// TIA Portal V20 export
FUNCTION_BLOCK "FB_Alarms_Safety"   // FB150, SCL
{ S7_Optimized_Access := 'TRUE' }
// stored: AutoNumber false, MemoryReserve 100, SetENOAutomatically false
   VAR
      sTimerEmergencyPowLaser : IEC_TIMER;
   END_VAR
BEGIN
   REGION Description header 
       //==================================================================================
       // POSALUX Swiss SA / (C) Copyright 2024
       //----------------------------------------------------------------------------------
       // Title: Affichage Alarmes/Messages Safety
       // Comment/Function: 
       //
       // Author: Michel FAIVRE
       // Engineering: TIA Portal v17
       //----------------------------------------------------------------------------------
       // Change log table:
       // Version  | Date     | Expert in charge | Changes applied
       // ---------|----------|------------------|------------------------------------
       // 01.01.00 | 20241218 | FMI              | First released version
       // ==================================================================================
   END_REGION

   REGION Warnings
       // Warning 700236 : Shutter ready to open, press laser button
       IF "LBP_AlarmMsgs".UserA[2].A70UUxx[36] AND
           ("MCP1_In".reset OR "DB_DataFromSafety".OpenShutter) THEN
           "LBP_AlarmMsgs".UserA[2].A70UUxx[36] := False;
       END_IF;
       IF NOT "LBP_AlarmMsgs".UserA[2].A70UUxx[36] AND NOT "DB_DataFromSafety".OpenShutter AND
           "DB_PowerOn".sMachinePower AND
           "DB_DataFromSafety".EmergencyStop AND
           "DB_DataFromSafety".iEmergencyStopPowerLaser AND
           "DB_DataFromSafety".iKeyLaserOn AND
           ("DB_DataFromSafety".iKeySettingLaser OR "DB_DataFromSafety".AllDoorLockedForLaser) THEN
           "LBP_AlarmMsgs".UserA[2].A70UUxx[36] := True;
       END_IF;

       // Warnings Doors
       "LBP_AlarmMsgs".UserA[5].A70UUxx[37] := NOT "DB_DataFromSafety".iFrontDoorClosed;
       "LBP_AlarmMsgs".UserA[5].A70UUxx[38] := NOT "DB_DataFromSafety".iMaintenanceDoorClosed;
       "LBP_AlarmMsgs".UserA[5].A70UUxx[39] := NOT "DB_DataFromSafety".iRoofLeftDoorClosed;
       "LBP_AlarmMsgs".UserA[5].A70UUxx[48] := NOT "DB_DataFromSafety".iRoofRightDoorClosed;

       // Warning 700542 : SAFETY : FEED STOP FOR ALL AXIS, MAIN DOOR IS CLOSED BUT NOT LOCKED
       IF "DB_DataFromSafety".iFrontDoorClosed
           AND NOT "DB_DigitalInputs".sFrontDoorLocked.sSWStatus  // Control Front Door locked
           AND "DB_DataFromSafety".iRoofLeftDoorClosed
           AND "DB_DataFromSafety".iRoofRightDoorClosed
           AND "DB_DataFromSafety".iKeySettingMode
           AND NOT "DB_McpKeyboardSignals".sAlarmReset.sKeySWStatus THEN
           IF "MCP1_In".minus OR "MCP1_In".plus THEN
               "LBP_AlarmMsgs".UserA[5].A70UUxx[42] := TRUE;
           END_IF;
       ELSE
           "LBP_AlarmMsgs".UserA[5].A70UUxx[42] := FALSE;
       END_IF;

       // Warning 700532 : SAFETY : COMMISSIONNING ON
       "LBP_AlarmMsgs".UserA[5].A70UUxx[32] := "DB_DataFromSafety".Comissionning;

       // Warning 700533 : SAFETY : LASER POWER SUPPLY IN EMERGENCY STOP
       #sTimerEmergencyPowLaser.TON(PT := t#200ms,
                                    IN := NOT "DB_DataFromSafety".iEmergencyStopPowerLaser);
       "LBP_AlarmMsgs".UserA[5].A70UUxx[33] := #sTimerEmergencyPowLaser.Q;

       // Warning 700534 : SAFETY : LASER SETTING MODE IS ACTIVE
       "LBP_AlarmMsgs".UserA[5].A70UUxx[34] := "DB_DataFromSafety".iKeySettingLaser;

       // Warning 700535 : SAFETY : LASER SHUTTER IS CLOSED
       "LBP_AlarmMsgs".UserA[5].A70UUxx[35] := "DB_DataFromSafety".ShutterClosed;

       // Warning 700536 : SAFETY : FEED STOP FOR ALL AXIS, PLEASE TURN SETTING KEY TO MOVE AXIS
       "LBP_AlarmMsgs".UserA[5].A70UUxx[36] := NOT "DB_DataFromSafety".DoorsClosed AND NOT "DB_DataFromSafety".iKeySettingMode;

       // Warning 700550 : SAFETY : KEY LASER OFF
       "LBP_AlarmMsgs".UserA[5].A70UUxx[50] := NOT "DB_DataFromSafety".iKeyLaserOn;

       // Warning 700551 : SAFETY : KEY LASER ON BUT LASER NOT READY
       "LBP_AlarmMsgs".UserA[5].A70UUxx[51] := "DB_DataFromSafety".iKeyLaserOn
       AND NOT "DB_DataFromSafety".ShutterReadyToOpen;

       // Warning 700552 : SAFETY : KEY LASER ON, LASER READY, SHUTTER CLOSED BY SOURCE
       // A implementer si l'entrée I0.7 SHUTTER IS CLOSED existe
       // "LBP_AlarmMsgs".UserA[5].A70UUxx[52] := "Main_Safety_RTG1_DB".SAFETY_LASER_KEY_ON
       // AND "Main_Safety_RTG1_DB".sLaserSupplyPower
       // AND "Main_Safety_RTG1_DB".SAFETY_EMERGENCY_STOP_POWER_LASER
       // AND (Shutter_is_closed) ;


   END_REGION

   REGION Alarms
       // Alarm 700500 : SAFETY : EMERGENCY STOP IS ACTIVE, PLEASE RESET  
       IF "DB_DataFromSafety".AckEmergencyStop THEN
           "LBP_AlarmMsgs".UserA[5].A70UUxx[0] := TRUE;
       END_IF;
       //  "LBP_AlarmMsgs".UserA[5].A70UUxx[0] := "DB_DataFromSafety".AckEmergencyStop;

       // Alarm 700501 : SAFETY : LASER POWER SUPPLY IS OFF, PLEASE RESET  
       IF NOT "DB_DataFromSafety".oContactorLaser THEN
           "LBP_AlarmMsgs".UserA[5].A70UUxx[1] := TRUE;
       END_IF;
       //   "LBP_AlarmMsgs".UserA[5].A70UUxx[1] := NOT "DB_DataFromSafety".oContactorLaser;

       // Alarm 700502 :SAFETY : LASER POWER SUPPLY IS NOT READY , PLEASE RESET
       IF NOT "DB_DataFromSafety".iEmergencyStopPowerLaser
           AND "DB_CycleStartStop".sChan1Start THEN
           "LBP_AlarmMsgs".UserA[5].A70UUxx[2] := TRUE;
       END_IF;

       // Alarm 700508 : SAFETY : FEEDBACK CONTACTOR POWER MACHINE IS NOT WORKING , PLEASE RESET
       IF "DB_DataFromSafety".SupplyPowerError AND "DB_PowerOn".sMachineReadySoft THEN
           "LBP_AlarmMsgs".UserA[5].A70UUxx[8] := TRUE;
       END_IF;

       // Alarm 700509 : SAFETY : FEEDBACK CONTACTOR POWER LASER IS NOT WORKING , PLEASE RESET
       IF "DB_DataFromSafety".LaserSupplyPowerError THEN
           "LBP_AlarmMsgs".UserA[5].A70UUxx[9] := TRUE;
       END_IF;

       // Alarm 700510 : SAFETY : FEEDBACK CONTACTOR OPEN SHUTTER IS NOT WORKING , PLEASE RESET
       IF "DB_DataFromSafety".ShutterError THEN
           "LBP_AlarmMsgs".UserA[5].A70UUxx[10] := TRUE;
       END_IF;

       // Alarm 700511 : SAFETY : FATAL ERROR ! : WRONG DISCORDANCE BEETWEEN SAFETY INPUTS, PLEASE RESET AND CHANGE SETTINGS
       "LBP_AlarmMsgs".UserA[5].A70UUxx[11] := "DB_DataFromSafety".AckI2001Functions;
   END_REGION
END_FUNCTION_BLOCK
